// TIA Portal V19 export
ORGANIZATION_BLOCK "Main"   // OB1, LAD, ProgramCycle
TITLE = "Main Program Sweep (Cycle)"
{ S7_Optimized_Access := 'TRUE' }
// stored: SetENOAutomatically false
   VAR_INPUT
      Initial_Call : Bool;   // Initial call of this OB
      Remanence : Bool;   // =True, if remanent data are available
   END_VAR
BEGIN

REGION Network 1: Dispenser
   // Running Code - Dispenser Project
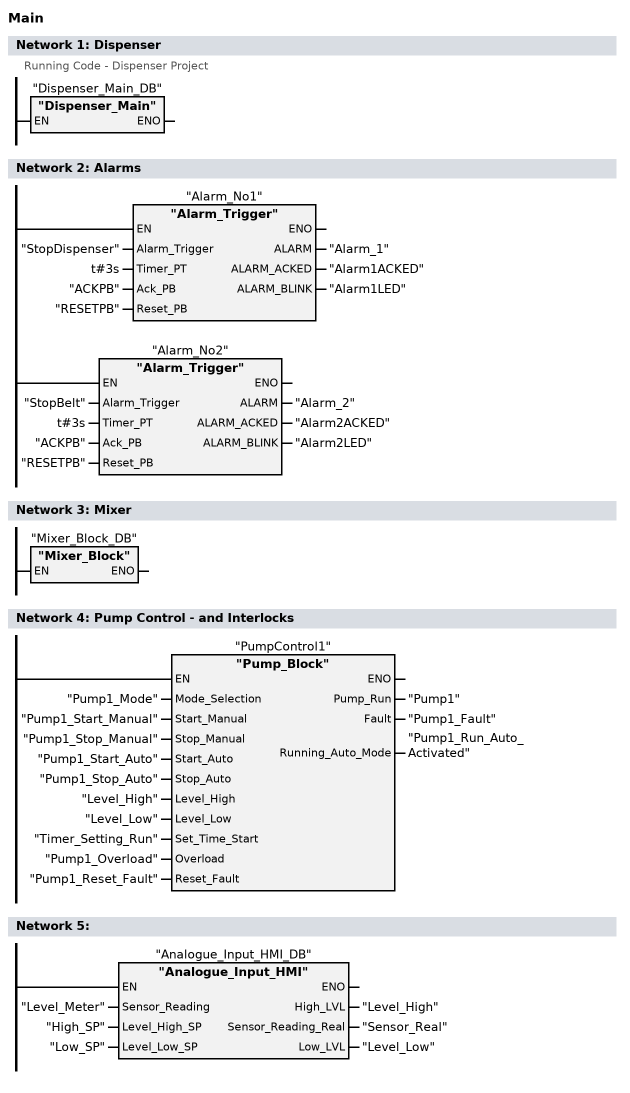
   RUNG wire#powerrail
      "Dispenser_Main_DB"()
   END_RUNG
   // the same network as SCL:
   "Dispenser_Main_DB"();   // "Dispenser_Main"
END_REGION

REGION Network 2: Alarms
   RUNG wire#powerrail
      "Alarm_No1"(Alarm_Trigger := "StopDispenser", Timer_PT := t#3s, Ack_PB := "ACKPB", Reset_PB := "RESETPB", ALARM => "Alarm_1", ALARM_ACKED => "Alarm1ACKED", ALARM_BLINK => "Alarm1LED")
   END_RUNG
   RUNG wire#powerrail
      "Alarm_No2"(Alarm_Trigger := "StopBelt", Timer_PT := t#3s, Ack_PB := "ACKPB", Reset_PB := "RESETPB", ALARM => "Alarm_2", ALARM_ACKED => "Alarm2ACKED", ALARM_BLINK => "Alarm2LED")
   END_RUNG
   // the same network as SCL:
   "Alarm_No1"(Alarm_Trigger := "StopDispenser",   // "Alarm_Trigger"
               Timer_PT := t#3s,
               Ack_PB := "ACKPB",
               Reset_PB := "RESETPB",
               ALARM => "Alarm_1",
               ALARM_ACKED => "Alarm1ACKED",
               ALARM_BLINK => "Alarm1LED");
   "Alarm_No2"(Alarm_Trigger := "StopBelt",   // "Alarm_Trigger"
               Timer_PT := t#3s,
               Ack_PB := "ACKPB",
               Reset_PB := "RESETPB",
               ALARM => "Alarm_2",
               ALARM_ACKED => "Alarm2ACKED",
               ALARM_BLINK => "Alarm2LED");
END_REGION

REGION Network 3: Mixer
   RUNG wire#powerrail
      "Mixer_Block_DB"()
   END_RUNG
   // the same network as SCL:
   "Mixer_Block_DB"();   // "Mixer_Block"
END_REGION

REGION Network 4: Pump Control - and Interlocks
   RUNG wire#powerrail
      "PumpControl1"(Mode_Selection := "Pump1_Mode", Start_Manual := "Pump1_Start_Manual", Stop_Manual := "Pump1_Stop_Manual", Start_Auto := "Pump1_Start_Auto", Stop_Auto := "Pump1_Stop_Auto", Level_High := "Level_High", Level_Low := "Level_Low", Set_Time_Start := "Timer_Setting_Run", Overload := "Pump1_Overload", Reset_Fault := "Pump1_Reset_Fault", Pump_Run => "Pump1", Fault => "Pump1_Fault", Running_Auto_Mode => "Pump1_Run_Auto_Activated")
   END_RUNG
   // the same network as SCL:
   "PumpControl1"(Mode_Selection := "Pump1_Mode",   // "Pump_Block"
                  Start_Manual := "Pump1_Start_Manual",
                  Stop_Manual := "Pump1_Stop_Manual",
                  Start_Auto := "Pump1_Start_Auto",
                  Stop_Auto := "Pump1_Stop_Auto",
                  Level_High := "Level_High",
                  Level_Low := "Level_Low",
                  Set_Time_Start := "Timer_Setting_Run",
                  Overload := "Pump1_Overload",
                  Reset_Fault := "Pump1_Reset_Fault",
                  Pump_Run => "Pump1",
                  Fault => "Pump1_Fault",
                  Running_Auto_Mode => "Pump1_Run_Auto_Activated");
END_REGION

REGION Network 5
   RUNG wire#powerrail
      "Analogue_Input_HMI_DB"(Sensor_Reading := "Level_Meter", Level_High_SP := "High_SP", Level_Low_SP := "Low_SP", High_LVL => "Level_High", Sensor_Reading_Real => "Sensor_Real", Low_LVL => "Level_Low")
   END_RUNG
   // the same network as SCL:
   "Analogue_Input_HMI_DB"(Sensor_Reading := "Level_Meter",   // "Analogue_Input_HMI"
                           Level_High_SP := "High_SP",
                           Level_Low_SP := "Low_SP",
                           High_LVL => "Level_High",
                           Sensor_Reading_Real => "Sensor_Real",
                           Low_LVL => "Level_Low");
END_REGION
END_ORGANIZATION_BLOCK
